FUNCTION_BLOCK Tank_StatusText IMPLEMENTS I_Call
VAR
	_ctx			: REFERENCE TO Tank_Ctx;
	_fbRec			: Receiver(THIS^);
END_VAR

METHOD Call
VAR_INPUT
	iTag	: Broadcast.Tags.I_Tag;
END_VAR
VAR
	cmp			: TagCmp;
END_VAR
cmp.Set(_ctx.priv.smgr.Current);			

IF cmp.Match(_ctx.state.iDisabled).IsOk() THEN
	_ctx.hmi.sStatusText := 'Tank disabled';
	_ctx.hmi.nStatusTextColor := COL.BLACK.Raw;
	RETURN;
END_IF

IF cmp.Match(_ctx.state.iEnabled).IsOk() THEN
	_ctx.hmi.sStatusText := 'Tank enabled';
	_ctx.hmi.nStatusTextColor := COL.BLACK.Raw;
	RETURN;
END_IF

IF cmp.Match(_ctx.state.iFault).IsOk() THEN
	_ctx.hmi.sStatusText := 'Alarm: Filling timeout!';
	_ctx.hmi.nStatusTextColor := COL.RED.Raw;
	RETURN;
END_IF

IF cmp.Match(_ctx.state.iFill).IsOk() THEN
	_ctx.hmi.sStatusText := 'Filling in progress...';
	_ctx.hmi.nStatusTextColor := COL.BLACK.Raw;
	RETURN;
END_IF

IF cmp.Match(_ctx.state.iSystemOff).IsOk() THEN
	_ctx.hmi.sStatusText := 'Filling system is disabled!';
	_ctx.hmi.nStatusTextColor := COL.BLACK.Raw;
	RETURN;
END_IF

IF cmp.Default() THEN
	_ctx.hmi.sStatusText := 'Error: Unrecognized system state.';
	_ctx.hmi.nStatusTextColor := COL.RED.Raw;
	RETURN;	
END_IF
END_METHOD

//FB_Init is always available implicitly and it is used primarily for initialization.
//The return value is not evaluated. For a specific influence, you can also declare the
//methods explicitly and provide additional code there with the standard initialization
//code. You can evaluate the return value.
METHOD FB_Init: BOOL
VAR_INPUT
    bInitRetains: BOOL; // TRUE: the retain variables are initialized (reset warm / reset cold)
    bInCopyCode: BOOL;  // TRUE: the instance will be copied to the copy code afterward (online change)
	
	ctx			: REFERENCE TO Tank_Ctx;
END_VAR
_ctx REF= ctx;
ctx.priv.smgr.GetOnChange().Pair(_fbRec);
END_METHOD

METHOD ToDebug : Debug.I_Debug
ToDebug := THIS^;
END_METHOD

END_FUNCTION_BLOCK

(* stored: Version 1.1.0.1
   POU Tank_StatusText: Id {fbdca127-14b9-4b94-8dc0-8bbde88ae7f1}, SpecialFunc None
   Method Call: Id {bc00e97c-e28d-4acb-88b7-451920d7a766}
   Method FB_init: Id {a9602e84-7aa2-4e0f-be51-20c49069a07b}
   Method ToDebug: Id {fd5b82b8-7e31-4600-bd43-1b0d6b9fa639} *)
